Fanuc KAREL source: SET_JPOS_TPE.kl

PROGRAM T
%NOLOCKGROUP
VAR
 v0 : INTEGER
 v1 : INTEGER
 v2 : JOINTPOS
 v3 : INTEGER
 v4 : INTEGER
BEGIN
 SET_JPOS_TPE(v0, v1, v2, v3, v4)
END T
